(* Logix 5000 project; controller SolisPLC_Vlad_CGL1 vendor 1 type 14 code 226 rev 36.11; software revision 36.00; part 2 of 3 *)
(* tags used below, declared in another part *)
   BOOL : BOOL[64];
   value : DINT;
   MQTT_OUT : UDT_MQTT_DINT[100];
   MQTT_OUT_BOOL : UDT_MQTT_DINT[100];
   MQTT_OUT_DINT : DINT[100];
   MTR1 : udtVariableSpeedMotor;
   MTR_Speed : REAL[100];
   Pal_D : DINT[100];
   Pal_T : TIMER[100];
   scanTime_G : DINT;
   ScanTimeMax : DINT;
   ScanTimeMin : DINT;
   Sys_Timer : TIMER[100];
   VFD_07 : udtVariableSpeedMotor;
(* Communication, continued *)

ROUTINE _03_VFD_Control   (* ladder *)
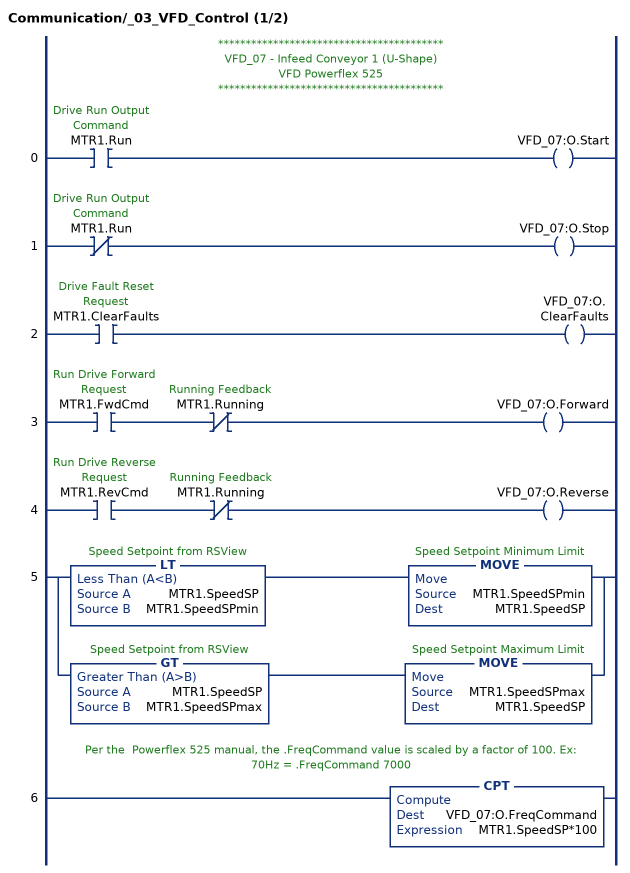
   // *****************************************
   // VFD_07 - Infeed Conveyor 1 (U-Shape)
   // VFD Powerflex 525
   // *****************************************
   0: XIC(MTR1.Run)OTE(VFD_07:O.Start);
   1: XIO(MTR1.Run)OTE(VFD_07:O.Stop);
   2: XIC(MTR1.ClearFaults)OTE(VFD_07:O.ClearFaults);
   3: XIC(MTR1.FwdCmd)XIO(MTR1.Running)OTE(VFD_07:O.Forward);
   4: XIC(MTR1.RevCmd)XIO(MTR1.Running)OTE(VFD_07:O.Reverse);
   5: [LT(MTR1.SpeedSP,MTR1.SpeedSPmin) MOVE(MTR1.SpeedSPmin,MTR1.SpeedSP) ,GT(MTR1.SpeedSP,MTR1.SpeedSPmax) MOVE(MTR1.SpeedSPmax,MTR1.SpeedSP) ];
   // Per the  Powerflex 525 manual, the .FreqCommand value is scaled by a factor of 100. Ex: 70Hz = .FreqCommand 7000
   6: CPT(VFD_07:O.FreqCommand,MTR1.SpeedSP*100);
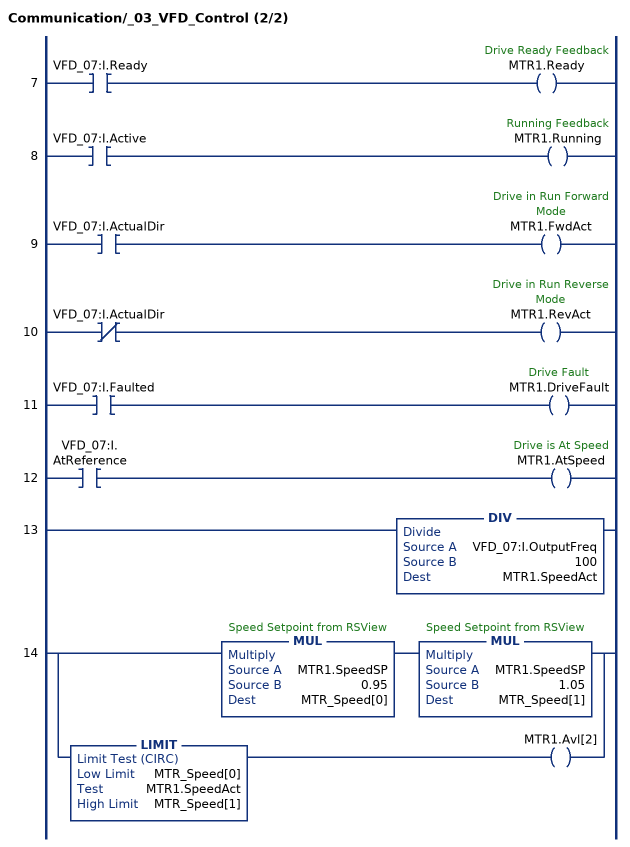
   7: XIC(VFD_07:I.Ready)OTE(MTR1.Ready);
   8: XIC(VFD_07:I.Active)OTE(MTR1.Running);
   9: XIC(VFD_07:I.ActualDir)OTE(MTR1.FwdAct);
   10: XIO(VFD_07:I.ActualDir)OTE(MTR1.RevAct);
   11: XIC(VFD_07:I.Faulted)OTE(MTR1.DriveFault);
   12: XIC(VFD_07:I.AtReference)OTE(MTR1.AtSpeed);
   13: DIV(VFD_07:I.OutputFreq,100,MTR1.SpeedAct);
   14: [MUL(MTR1.SpeedSP,0.95,MTR_Speed[0]) MUL(MTR1.SpeedSP,1.05,MTR_Speed[1]) ,LIMIT(MTR_Speed[0],MTR1.SpeedAct,MTR_Speed[1]) OTE(MTR1.Avl[2]) ];
END_ROUTINE
END_PROGRAM

PROGRAM DataLink   (* main routine _01_Main *)
VAR
   index : DINT := 100;
END_VAR

ROUTINE _01_Main   (* ladder *)
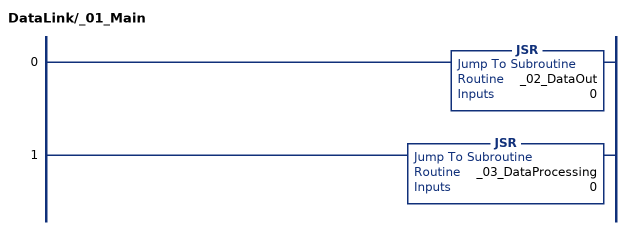
   0: JSR(_02_DataOut,0);
   1: JSR(_03_DataProcessing,0);
END_ROUTINE

ROUTINE _02_DataOut   (* ladder *)
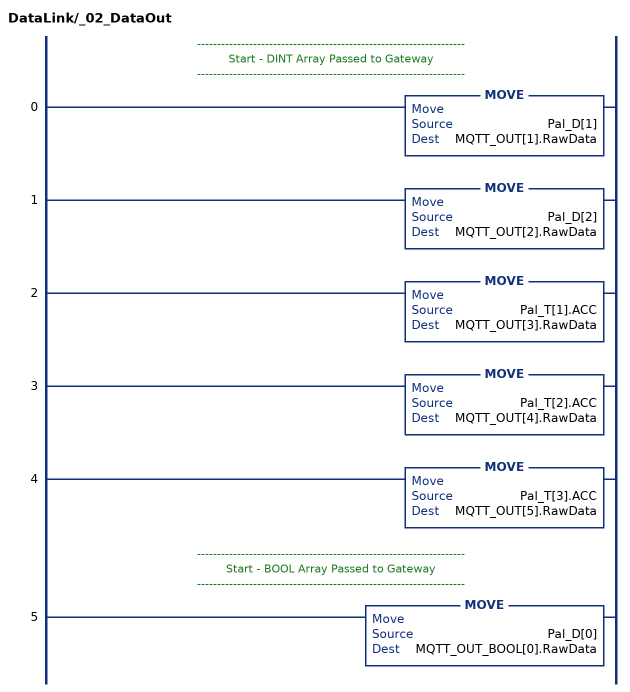
   // -------------------------------------------------------------------
   // Start - DINT Array Passed to Gateway
   // -------------------------------------------------------------------
   0: MOVE(Pal_D[1],MQTT_OUT[1].RawData);
   1: MOVE(Pal_D[2],MQTT_OUT[2].RawData);
   2: MOVE(Pal_T[1].ACC,MQTT_OUT[3].RawData);
   3: MOVE(Pal_T[2].ACC,MQTT_OUT[4].RawData);
   4: MOVE(Pal_T[3].ACC,MQTT_OUT[5].RawData);
   // -------------------------------------------------------------------
   // Start - BOOL Array Passed to Gateway
   // -------------------------------------------------------------------
   5: MOVE(Pal_D[0],MQTT_OUT_BOOL[0].RawData);
END_ROUTINE

ROUTINE _03_DataProcessing   (* ladder *)
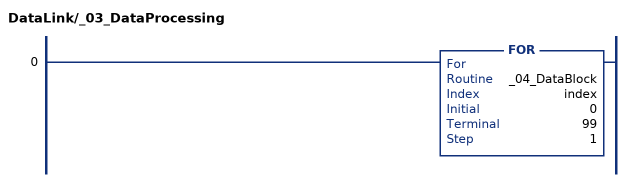
   0: FOR(_04_DataBlock,index,0,99,1);
END_ROUTINE

ROUTINE _04_DataBlock   (* ladder *)
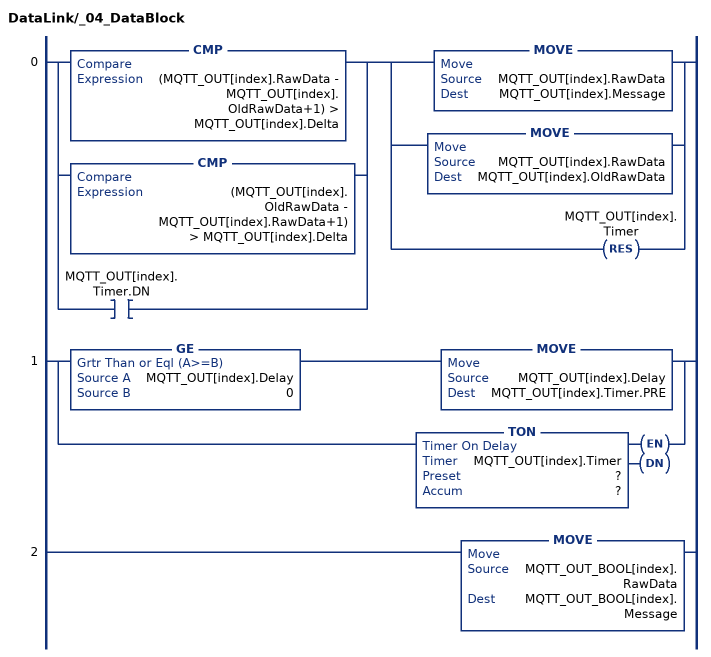
   0: [CMP((MQTT_OUT[index].RawData - MQTT_OUT[index].OldRawData+1) > MQTT_OUT[index].Delta) ,CMP((MQTT_OUT[index].OldRawData - MQTT_OUT[index].RawData+1) > MQTT_OUT[index].Delta) ,XIC(MQTT_OUT[index].Timer.DN) ][MOVE(MQTT_OUT[index].RawData,MQTT_OUT[index].Message) ,MOVE(MQTT_OUT[index].RawData,MQTT_OUT[index].OldRawData) ,RES(MQTT_OUT[index].Timer) ];
   1: [GE(MQTT_OUT[index].Delay,0) MOVE(MQTT_OUT[index].Delay,MQTT_OUT[index].Timer.PRE) ,TON(MQTT_OUT[index].Timer,?,?) ];
   2: MOVE(MQTT_OUT_BOOL[index].RawData,MQTT_OUT_BOOL[index].Message);
END_ROUTINE
END_PROGRAM

PROGRAM MainProgram   (* main routine MainRoutine *)

ROUTINE MainRoutine   (* ladder *)
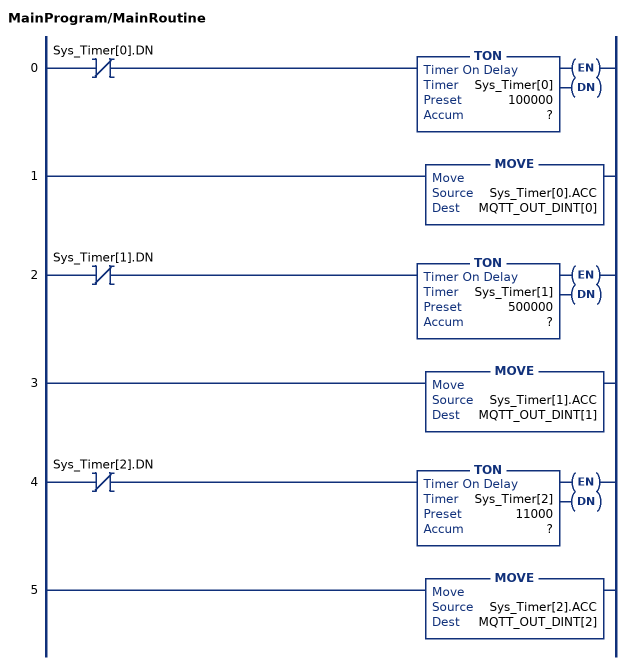
   0: XIO(Sys_Timer[0].DN)TON(Sys_Timer[0],?,?);
   1: MOVE(Sys_Timer[0].ACC,MQTT_OUT_DINT[0]);
   2: XIO(Sys_Timer[1].DN)TON(Sys_Timer[1],?,?);
   3: MOVE(Sys_Timer[1].ACC,MQTT_OUT_DINT[1]);
   4: XIO(Sys_Timer[2].DN)TON(Sys_Timer[2],?,?);
   5: MOVE(Sys_Timer[2].ACC,MQTT_OUT_DINT[2]);
END_ROUTINE
END_PROGRAM

PROGRAM Palletizer   (* main routine _01_Main *)
VAR
   Mask : DINT[20];
   Mask1 : DINT;
   NumberofCasesAtInfeed : DINT := 9;
   Pal_ONS : BOOL[64] := ([0] := 1);
   RandomNum : DINT := 51666400;
   ScanTime : DINT := 233;
   SystemFaulted : BOOL;
   SystemIdle : BOOL;
   SystemRunning : BOOL;
   SystemStatus : DINT;
   Time : DINT[7] := ([0] := 1998, [1] := 5, [2] := 10, [3] := 18, [4] := 10, [5] := 15, [6] := 886159);
END_VAR

ROUTINE _01_Main   (* ladder *)
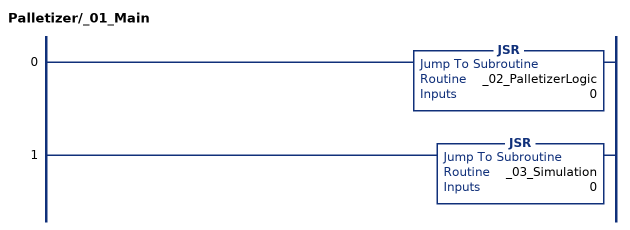
   0: JSR(_02_PalletizerLogic,0);
   1: JSR(_03_Simulation,0);
END_ROUTINE

ROUTINE _02_PalletizerLogic   (* ladder *)
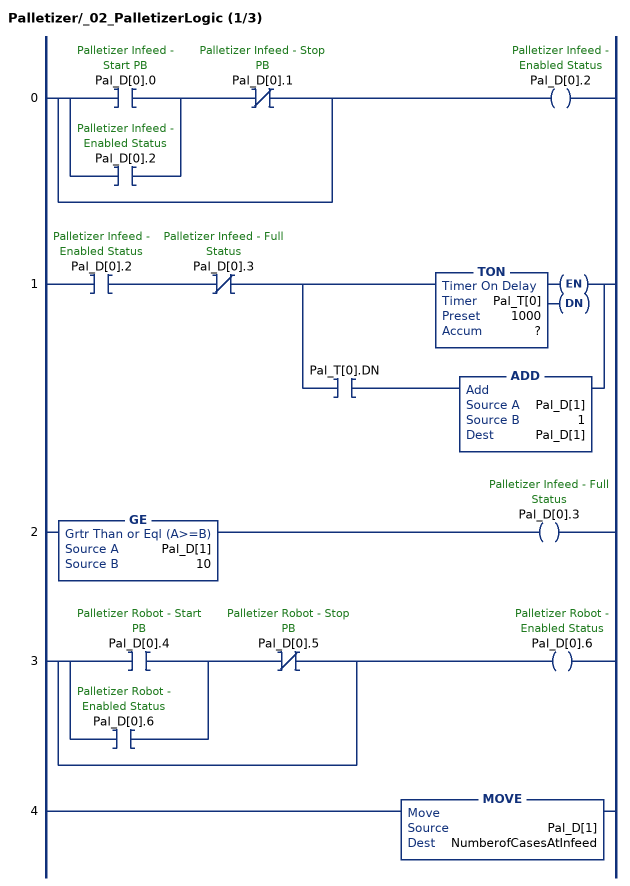
   0: [[XIC(Pal_D[0].0) ,XIC(Pal_D[0].2) ] XIO(Pal_D[0].1) ,]OTE(Pal_D[0].2);
   1: XIC(Pal_D[0].2)XIO(Pal_D[0].3)[TON(Pal_T[0],?,?) ,XIC(Pal_T[0].DN) ADD(Pal_D[1],1,Pal_D[1]) ];
   2: GE(Pal_D[1],10)OTE(Pal_D[0].3);
   3: [[XIC(Pal_D[0].4) ,XIC(Pal_D[0].6) ] XIO(Pal_D[0].5) ,]OTE(Pal_D[0].6);
   4: MOVE(Pal_D[1],NumberofCasesAtInfeed);
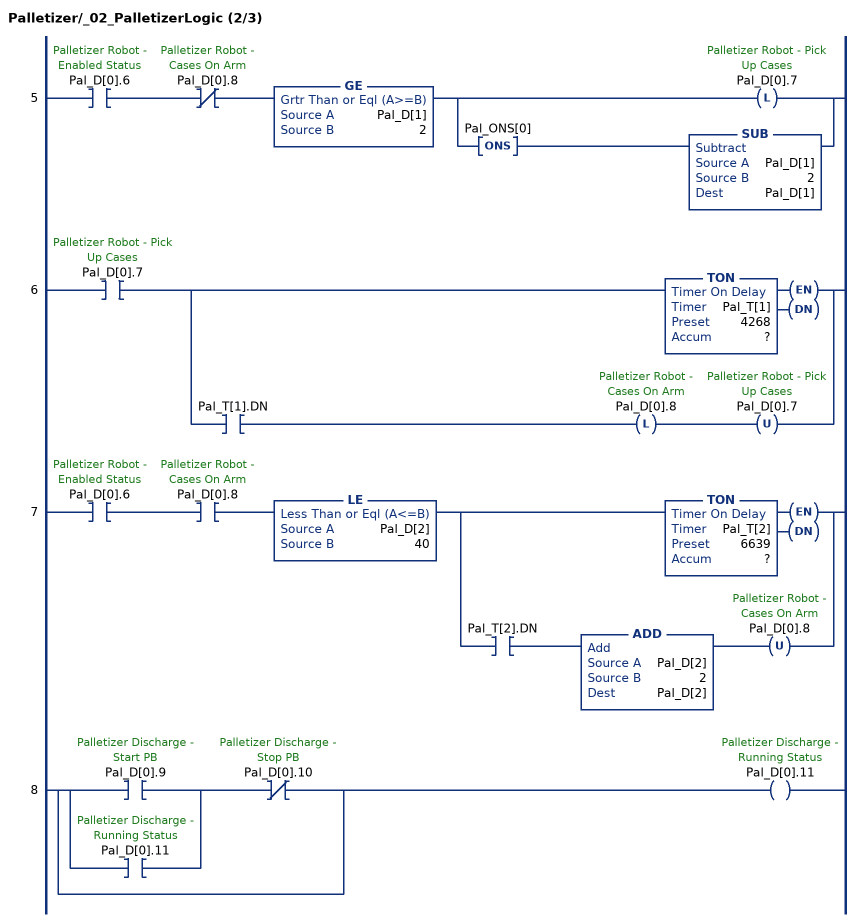
   5: XIC(Pal_D[0].6)XIO(Pal_D[0].8)GE(Pal_D[1],2)[OTL(Pal_D[0].7) ,ONS(Pal_ONS[0]) SUB(Pal_D[1],2,Pal_D[1]) ];
   6: XIC(Pal_D[0].7)[TON(Pal_T[1],?,?) ,XIC(Pal_T[1].DN) OTL(Pal_D[0].8) OTU(Pal_D[0].7) ];
   7: XIC(Pal_D[0].6)XIC(Pal_D[0].8)LE(Pal_D[2],40)[TON(Pal_T[2],?,?) ,XIC(Pal_T[2].DN) ADD(Pal_D[2],2,Pal_D[2]) OTU(Pal_D[0].8) ];
   8: [[XIC(Pal_D[0].9) ,XIC(Pal_D[0].11) ] XIO(Pal_D[0].10) ,]OTE(Pal_D[0].11);
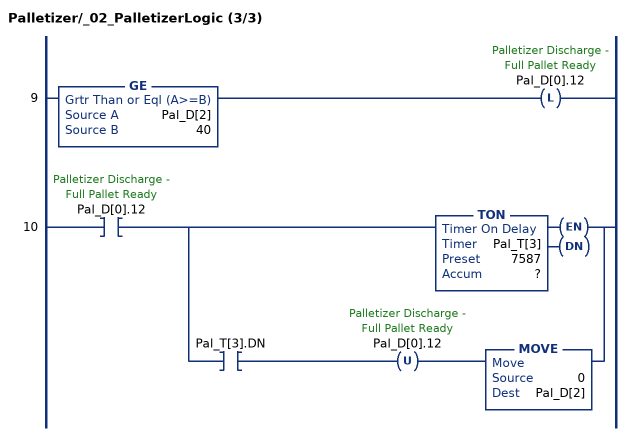
   9: GE(Pal_D[2],40)OTL(Pal_D[0].12);
   10: XIC(Pal_D[0].12)[TON(Pal_T[3],?,?) ,XIC(Pal_T[3].DN) OTU(Pal_D[0].12) MOVE(0,Pal_D[2]) ];
END_ROUTINE

ROUTINE _03_Simulation   (* ladder *)
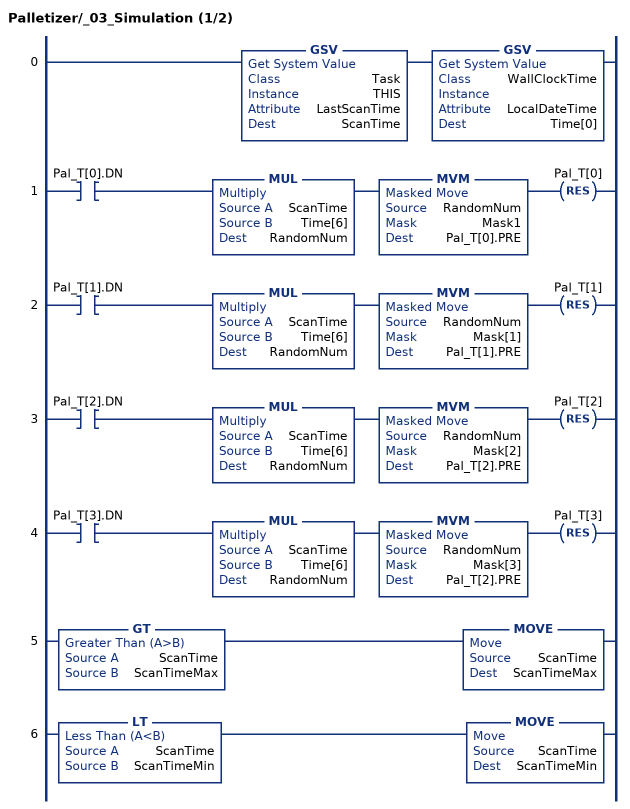
   0: GSV(Task,THIS,LastScanTime,ScanTime)GSV(WallClockTime,,LocalDateTime,Time[0]);
   1: XIC(Pal_T[0].DN)MUL(ScanTime,Time[6],RandomNum)MVM(RandomNum,Mask1,Pal_T[0].PRE)RES(Pal_T[0]);
   2: XIC(Pal_T[1].DN)MUL(ScanTime,Time[6],RandomNum)MVM(RandomNum,Mask[1],Pal_T[1].PRE)RES(Pal_T[1]);
   3: XIC(Pal_T[2].DN)MUL(ScanTime,Time[6],RandomNum)MVM(RandomNum,Mask[2],Pal_T[2].PRE)RES(Pal_T[2]);
   4: XIC(Pal_T[3].DN)MUL(ScanTime,Time[6],RandomNum)MVM(RandomNum,Mask[3],Pal_T[2].PRE)RES(Pal_T[3]);
   5: GT(ScanTime,ScanTimeMax)MOVE(ScanTime,ScanTimeMax);
   6: LT(ScanTime,ScanTimeMin)MOVE(ScanTime,ScanTimeMin);
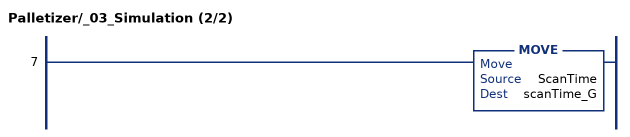
   7: MOVE(ScanTime,scanTime_G);
END_ROUTINE
END_PROGRAM

PROGRAM SafetyProgram   (* main routine MainRoutine, safety *)

ROUTINE MainRoutine   (* ladder *)
END_ROUTINE
END_PROGRAM

PROGRAM SimulatedMachine_v1_0   (* main routine _01_Main *)
VAR
   Mach_ControlDINT : DINT[10] := ([0] := 16, [1] := 466);
        [0].0   // Machine Start
        [0].1   // Machine Stop
        [0].2   // Machine State - Running
        [0].3   // Machine - Making a Part!
   Mach_ControlTIMER : TIMER[100] := ([0].PRE := 1867);
   Mach_DataDINT : DINT[100] := ([1] := 13, [2] := 1);
   Mach_SimDINT : DINT[100] := ([0] := 15, [1] := 374, [2] := 54000000, [4] := 50000, [5] := 750000);
   Mach_SimREAL : REAL[100] := ([0] := 144385.03, [1] := 2005.3475);
   Mach_SimTIMER : TIMER[100] := ([0].PRE := 154424);
END_VAR

ROUTINE _01_Main   (* ladder *)
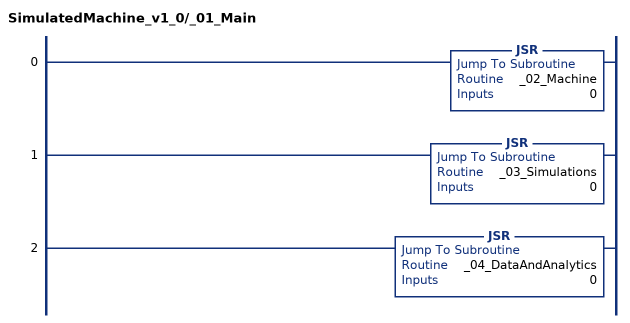
   0: JSR(_02_Machine,0);
   1: JSR(_03_Simulations,0);
   2: JSR(_04_DataAndAnalytics,0);
END_ROUTINE

ROUTINE _02_Machine   (* ladder *)
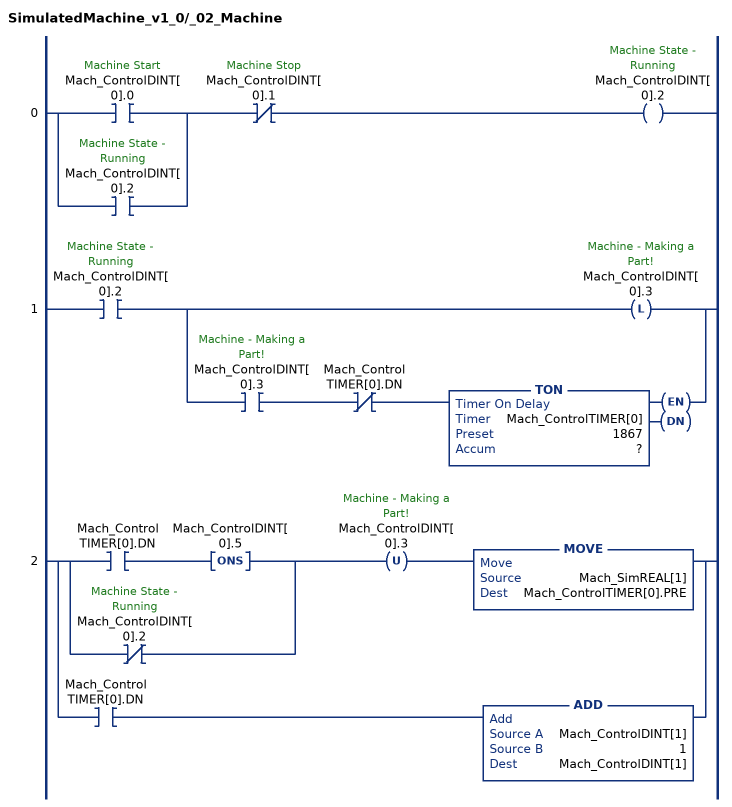
   0: [XIC(Mach_ControlDINT[0].0) ,XIC(Mach_ControlDINT[0].2) ]XIO(Mach_ControlDINT[0].1)OTE(Mach_ControlDINT[0].2);
   1: XIC(Mach_ControlDINT[0].2)[OTL(Mach_ControlDINT[0].3) ,XIC(Mach_ControlDINT[0].3) XIO(Mach_ControlTIMER[0].DN) TON(Mach_ControlTIMER[0],?,?) ];
   2: [[XIC(Mach_ControlTIMER[0].DN) ONS(Mach_ControlDINT[0].5) ,XIO(Mach_ControlDINT[0].2) ] OTU(Mach_ControlDINT[0].3) MOVE(Mach_SimREAL[1],Mach_ControlTIMER[0].PRE) ,XIC(Mach_ControlTIMER[0].DN) ADD(Mach_ControlDINT[1],1,Mach_ControlDINT[1]) ];
END_ROUTINE

ROUTINE _03_Simulations   (* ladder *)
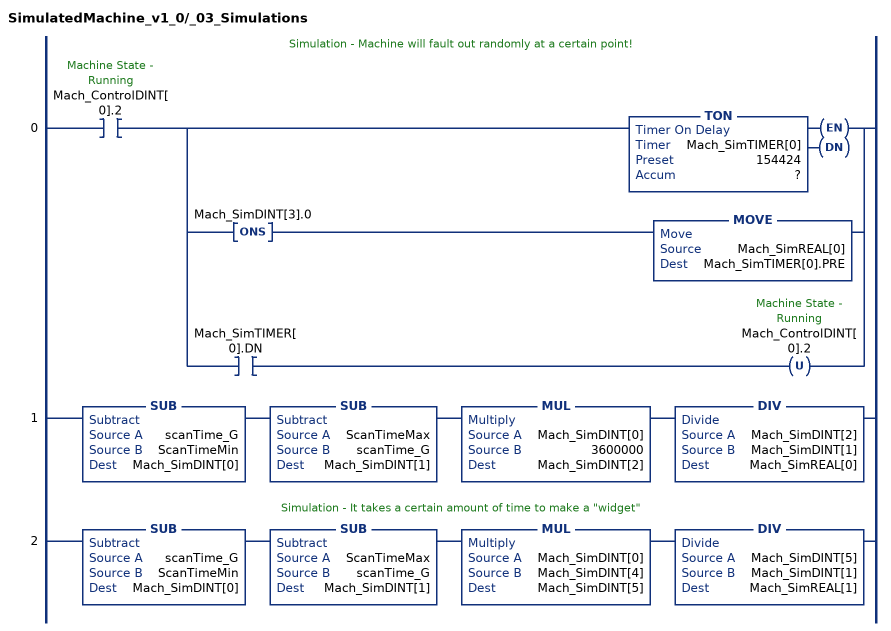
   // Simulation - Machine will fault out randomly at a certain point!
   0: XIC(Mach_ControlDINT[0].2)[TON(Mach_SimTIMER[0],?,?) ,ONS(Mach_SimDINT[3].0) MOVE(Mach_SimREAL[0],Mach_SimTIMER[0].PRE) ,XIC(Mach_SimTIMER[0].DN) OTU(Mach_ControlDINT[0].2) ];
   1: SUB(scanTime_G,ScanTimeMin,Mach_SimDINT[0])SUB(ScanTimeMax,scanTime_G,Mach_SimDINT[1])MUL(Mach_SimDINT[0],3600000,Mach_SimDINT[2])DIV(Mach_SimDINT[2],Mach_SimDINT[1],Mach_SimREAL[0]);
   // Simulation - It takes a certain amount of time to make a "widget"
   2: SUB(scanTime_G,ScanTimeMin,Mach_SimDINT[0])SUB(ScanTimeMax,scanTime_G,Mach_SimDINT[1])MUL(Mach_SimDINT[0],Mach_SimDINT[4],Mach_SimDINT[5])DIV(Mach_SimDINT[5],Mach_SimDINT[1],Mach_SimREAL[1]);
END_ROUTINE

ROUTINE _04_DataAndAnalytics   (* ladder *)
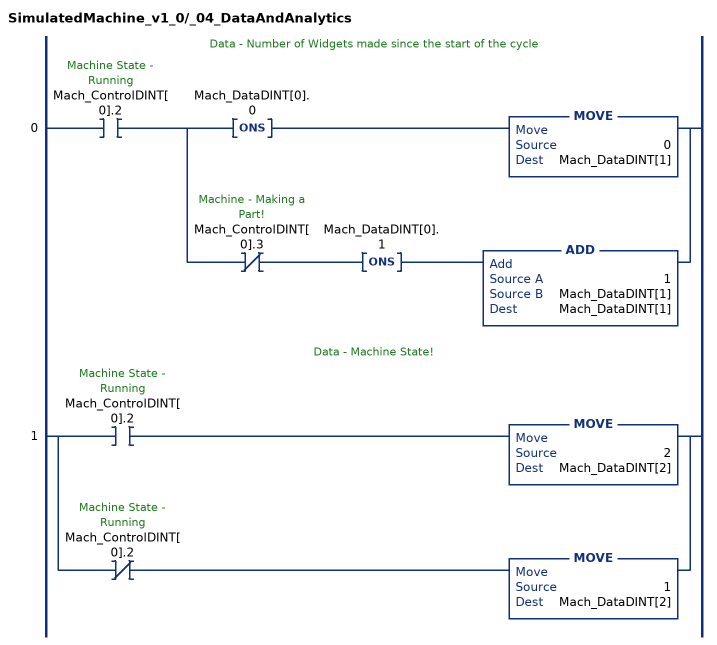
   // Data - Number of Widgets made since the start of the cycle
   0: XIC(Mach_ControlDINT[0].2)[ONS(Mach_DataDINT[0].0) MOVE(0,Mach_DataDINT[1]) ,XIO(Mach_ControlDINT[0].3) ONS(Mach_DataDINT[0].1) ADD(1,Mach_DataDINT[1],Mach_DataDINT[1]) ];
   // Data - Machine State!
   1: [XIC(Mach_ControlDINT[0].2) MOVE(2,Mach_DataDINT[2]) ,XIO(Mach_ControlDINT[0].2) MOVE(1,Mach_DataDINT[2]) ];
END_ROUTINE
END_PROGRAM

PROGRAM Tutorials   (* main routine _01_Main *)
VAR
   _AOI_Fah_to_Cel1 : _AOI_Fah_to_Cel := (Temperature_Fah := 100.0, Temperature_Cel := 37.77778);
   _AOI_Fah_to_Cel2 : _AOI_Fah_to_Cel := (Temperature_Cel := -17.777779);
   BoxID : DINT := 3333;
   BoxRejectSystem : DINT[100] := ([0] := 2222, [1] := 2222, [2] := 2222, [3] := 2222, [4] := 3333, [5] := 3333);
   BoxRejectSystem_CTRL : CONTROL := (LEN := 100, POS := 6);
   CasePackerBackUpTimer : TIMER := (PRE := 3000);
   Conv1_Disch_BoxCounter : COUNTER := (ACC := 513, DN := 1);
   MC_Running : BOOL;
   MCO_T1 : TIMER := (PRE := 5000);
   MCO_T10 : TIMER := (PRE := 2000);
   MCO_T11 : TIMER := (PRE := 2000);
   MCO_T2 : TIMER := (PRE := 5000);
   MCO_T3 : TIMER := (PRE := 3000);
   MCO_T4 : TIMER := (PRE := 1000);
   MCO_T5 : TIMER := (PRE := 3000);
   MCO_T6 : TIMER := (PRE := 3000);
   MCO_T7 : TIMER;
   MCO_T8 : TIMER := (PRE := 2000);
   MCO_T9 : TIMER := (PRE := 1000);
   NarrowBox_Counter : COUNTER := (ACC := 22, DN := 1);
   NarrowBox_CTU : COUNTER := (ACC := 201, DN := 1);
   PalletizerEMptyTimer : TIMER := (PRE := 10000, ACC := 10000, EN := 1, DN := 1);
   PalletizerNeedsCase : BOOL := 1;
   PartAssemblySeqStep : DINT;
   Placeholder1 : REAL := -32.0;
   Placeholder2 : REAL := -160.0;
   RejectID : DINT := 2222;
   S2_CasePackerBackedUp : BOOL;
   S2_Output : BOOL;
   S2_Output1 : BOOL;
   S2_PalletizerBoxAtInfeedSensor : BOOL;
   S2_PalletizerCaseInside : BOOL;
   S2_PalletizerCaseInside2 : BOOL;
   S2_Storage : BOOL;
   S2_Storage1 : BOOL;
   S2_SystemRunning : BOOL;
   SCADA_ProduceLids : BOOL := 1;
   SolisPLC_ONS : BOOL[64];
   TempC1 : REAL := -17.777779;
   TempC2 : REAL := 37.77778;
   TempC3 : REAL := -17.777779;
   TempF1 : REAL;
   TempF2 : REAL := 100.0;
   TempF3 : REAL;
   Test_CaseID : DINT := 4444;
   Test_FIFO_CaseReject : DINT[100] := ([0] := 4444, [1] := 4444, [2] := 4444, [3] := 3333, [4] := 4444, [5] := 3333, [6] := 3333, [7] := 4444, [8] := 3333, [9] := 3333, [10] := 3333, [11] := 4444, [12] := 4444, [13] := 3333, [14] := 3333, [15] := 3333, [16] := 4444, [17] := 3333, [18] := 4444, [19] := 4444, [20] := 3333, [21] := 4444);
   Test_FIFO_CaseRejectCTRL : CONTROL := (LEN := 50, POS := 22);
   Test_FIFO_CaseState : DINT := 3333;
   WideBoc_CTU : COUNTER;
   WideBox_Counter : COUNTER := (DN := 1);
   WideBox_CTU : COUNTER := (ACC := 183, DN := 1);
END_VAR

ROUTINE _01_Main   (* ladder *)
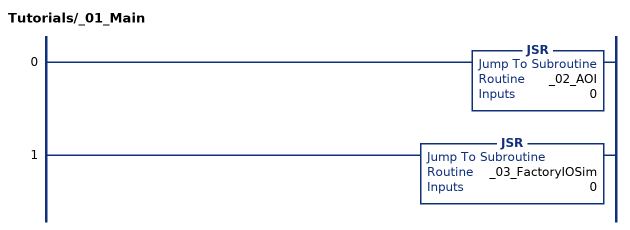
   0: JSR(_02_AOI,0);
   1: JSR(_03_FactoryIOSim,0);
END_ROUTINE
